// TIA Portal V17 export
// export: Created 2024-09-02T12:50:04.8053411Z, ExportSetting WithDefaults, DisplayName Totally Integrated Automation Portal, DisplayVersion V17, DisplayName TIA Portal Openness, DisplayVersion V17, DisplayName TIA Portal Version Control Interface, DisplayVersion V17, DisplayName STEP 7 Professional, DisplayVersion V17, DisplayName STEP 7 Safety, DisplayVersion V17, DisplayName WinCC Professional, DisplayVersion V17
DATA_BLOCK "AnwDB_Finished"   // DB181
{ S7_Optimized_Access := 'TRUE'; DB_Accessible_From_OPC_UA := 'FALSE' }
VERSION : 0.1
// stored: AutoNumber false, DBAccessibleFromOPCUA false, IsOnlyStoredInLoadMemory false, IsRetainMemResEnabled false, IsWriteProtectedInAS false, MemoryReserve 1000
   VAR RETAIN
      OP70_1 { ExternalWritable := 'False'} : Struct   // FG
         Finished { ExternalWritable := 'False'} : Bool;   // Anwender Fertigmeldung / User finish message
      END_STRUCT;
      OP70_2 { ExternalWritable := 'False'} : Struct   // FG
         Finished { ExternalWritable := 'False'} : Bool;   // Anwender Fertigmeldung / User finish message
      END_STRUCT;
   END_VAR
BEGIN
END_DATA_BLOCK
